FUNCTION_BLOCK FB_SmartGripper EXTENDS GrundstrukturObjekt
VAR_INPUT
	sIP					:T_IPv4Addr;
	iPort				:UINT;
END_VAR
VAR_OUTPUT
	
END_VAR
VAR
	// Instanziierung von Kommunikationsbausteine
	Communication_send		:ModbusRtuMasterV2_PcCOM;
	Communication_receive	:ModbusRtuMasterV2_PcCOM;
	
	// Kommunikationsvariablen
	UnitID      		:BYTE := 9;
    Quantity    		:WORD := 1;
    MBAddr      		:WORD := 16#1000;
    Execute     		:BOOL;
    Timeout     		:TIME := T#5S;
	
	cbRead				:UINT;
	State				:INT;
	
	
	Senddaten 			:ARRAY[0..15] OF BYTE;
	TEST				:TEST;

	
	Modbusdaten: BYTE;
END_VAR



// Instanziierungen
Senddaten[0] := 9;
Senddaten[1] := 16;
Senddaten[2] := 3;
Senddaten[3] := 232;
Senddaten[4] := 0;
Senddaten[5] := 3;
Senddaten[6] := 6;
Senddaten[7] := 0;
Senddaten[8] := 0;
Senddaten[9] := 0;
Senddaten[10] := 0;
Senddaten[11] := 0;
Senddaten[12] := 0; 
Senddaten[13] := 115;
Senddaten[14] := 48;
Senddaten[15] := 0;	
			
TEST.arrByte := Senddaten;

//Communication_§end.WriteSingleRegister();
Communication_send.WriteSingleRegister(UnitID := UnitID,
										Quantity := Quantity,
										MBAddr := MBAddr,
										cbLength := SIZEOF(Senddaten),
										pMemoryAddr := ADR(Senddaten),
										Execute := Execute,
										Timeout := Timeout,
										BUSY => bBusy,
										Error => bError,
										ErrorId => iErrorID,
										cbRead => cbRead);
				

//____________________________________________________________________________________________
// Input-Command-Verwaltung

//____________________________________________________________________________________________
// Interner Methodenaufruf (Durch System oder Skill)

//____________________________________________________________________________________________
// Datenerfassungsprozess

//____________________________________________________________________________________________
// Zustandsmanagement

	CASE iState OF 
		0: // AUS
			// DO
		
			// TRANSITION
		
		//____________________________________________________________________________________________
		1: // BEREIT
			// DO

			// TRANSITION
		
		//____________________________________________________________________________________________
		2: // MANUELL
			// DO
		
			// TRANSITION
		
		//____________________________________________________________________________________________
		3: // LAUFEND
			// DO
		
			// TRANSITION
		
		//____________________________________________________________________________________________
		4: // ABGESCHLOSSEN
			// DO
		
			// TRANSITION
		
		//____________________________________________________________________________________________
		5: // GESTOPPT
			// DO
		
			// TRANSITION
		
		//____________________________________________________________________________________________
		6: // FEHLER
			// DO
		
			// TRANSITION
		
		
	END_CASE

METHOD DoSomething : BOOL
VAR_INPUT
	
END_VAR
VAR
	
END_VAR
END_METHOD

METHOD Trennen : BOOL
VAR_INPUT
END_VAR
END_METHOD

METHOD Verbinden : BOOL
VAR_INPUT
END_VAR
END_METHOD

END_FUNCTION_BLOCK

(* stored: Version 1.1.0.1
   POU FB_SmartGripper: Id {35840996-72e9-4e57-ab7f-da4985d9fd20}, SpecialFunc None
   Folder 01_Methoden: Id {7d669dd2-3272-4c05-9652-b24101f6a60c}
   Folder 01_Nicht_Funktional: Id {ad9c4ca0-e515-4ee4-b2d1-299ee97cb244}
   Folder 02_Funktional: Id {b676063b-86a0-4d98-9f10-67cb64c180e0}
   Folder 02_Eigenschaften: Id {06046150-532d-40ac-ab56-fa8157a0bff3}
   Method DoSomething: Id {866858fa-1fed-4bb7-8ac4-4ce20c82c07d}
   Method Trennen: Id {cfb8b5e8-647a-492b-85b8-243233eaa6b0}
   Method Verbinden: Id {dd15742f-3230-453e-96b7-d7eeac293a9d} *)
